{attribute 'qualified_only'}
VAR_GLOBAL
	HMI_CNV_SftyPinDown_1:  BOOL;
	HMI_CNV_SftyPinUp_1:  BOOL;
	HMI_Light_Guard:  Bool;
	HMI_CNV_Forward_1:  Bool;
	HMI_CNV_Backward:  Bool;
	HMI_CNV_Forward:  Bool;
	HMI_CNV_Backward_1:  Bool;
END_VAR

(* stored: Version 1.1.0.1
   GVL CNV_HMI_IO: Id {986cc9d9-1172-4de4-8901-003e30101265} *)
